FUNCTION_BLOCK FB_HydMixCirc
VAR_INPUT
	iPump			:	I_Pump;
	iValve			:	I_Valve;
	iTempSupPrim	:	I_TempSens;
	iTempRetPrim	:	I_TempSens;
	iTempSup		:	I_TempSens;
	iTempRet		:	I_TempSens;
	iControl		:	I_HydMixCircControl;
	eModeSet 		:	E_ControlMode := E_ControlMode.Off;	// set control mode
	bInit			:	BOOL;
END_VAR
VAR_OUTPUT
	bErr	:	BOOL;
END_VAR
VAR	
END_VAR

//Update temperatures
iTempSupPrim.Run();
iTempRetPrim.Run();
iTempSup.Run();
iTempRet.Run();

//Run Controller
IF bInit THEN
	iControl.TempAct := iTempSup.Temperature;
	iControl.Init();
ELSE
	iControl.ModeSet := eModeSet; //Mode setpoint
	iControl.TempAct := iTempSup.Temperature;
	iControl.Run();
END_IF
	
//Pump
iPump.Setpoint := iControl.PumpSet;
iPump.SetOn := TRUE;
iPump.ControlMode := iControl.PumpMode;

//Valve
iValve.OpenPercSet := iControl.ValveSet;

//Run components
iPump.Run();
iValve.Run();

IF iPump.Error OR iValve.Error OR iControl.Error THEN
	bErr := TRUE;
ELSE
	bErr := FALSE;
END_IF

END_FUNCTION_BLOCK

(* stored: Version 1.1.0.1, ProductVersion 3.1.4022.10
   POU FB_HydMixCirc: Id {eabd025c-8904-4613-9374-1385642bd5cf}, SpecialFunc None *)
